// TIA Portal V19 export
VAR_GLOBAL   // PLC tag table "Default tag table"
   "CPU RUN" AT %I0.0 : Bool;
   "SPARE(1)" AT %I0.1 : Bool;
   "SPARE(2)" AT %I0.2 : Bool;
   "P-201 A RO 1 FEED PUMP TRIP" AT %I0.3 : Bool;
   "P-201 B RO 1 FEED PUMP TRIP" AT %I0.4 : Bool;
   "P-201 C RO 1 FEED PUMP TRIP" AT %I0.5 : Bool;
   "P-301 A RO 1 HPP PUMP TRIP" AT %I0.6 : Bool;
   "P-301 B RO B HPP PUMP TRIP" AT %I0.7 : Bool;
   "P-401 A RO 2 FEED PUMP TRIP" AT %I1.0 : Bool;
   "P-401 B RO 2 FEED PUMP TRIP" AT %I1.1 : Bool;
   "P-401 C RO 2 FEED PUMP TRIP" AT %I1.2 : Bool;
   "P 401 A RO 2 HPP PUMP TRIP" AT %I1.3 : Bool;
   "P-401 B RO 2 HPP PUMP TRIP" AT %I1.4 : Bool;
   "LPS 301 RO 1" AT %I1.5 : Bool;
   "P-202 A RO 1 FEED PUMP" AT %Q0.0 : Bool;
   "P-202 B RO 1 FEED PUMP" AT %Q0.1 : Bool;
   "P-202 C RO 1 FEED PUMP" AT %Q0.2 : Bool;
   "P-301 A RO 1 HPP PUMP" AT %Q0.3 : Bool;
   "P-301 B RO 1 HPP PUMP" AT %Q0.4 : Bool;
   "P-401 A RO 2 FEED PUMP" AT %Q0.5 : Bool;
   "P-401 B RO 2 FEED PUMP" AT %Q0.6 : Bool;
   "P-401 C RO 2 FEED PUMP" AT %Q0.7 : Bool;
   "P-402  A RO 2 HPP" AT %Q1.0 : Bool;
   "P-402 B" AT %Q1.1 : Bool;
   "HPS-301 RO 1 PRESSURE SWITCH" AT %I8.0 : Bool;
   "LPS-302 RO 1 PRESSURE SWITCH" AT %I8.1 : Bool;
   "HPS-302 RO 1 PRESSURE SWITCH" AT %I8.2 : Bool;
   "LPS-401 RO 2 PRESSURE SWITCH" AT %I8.3 : Bool;
   "HPS-401 RO 2 PRESSURE SWITCH" AT %I8.4 : Bool;
   "LPS-402 RO 2 PRESSURE SWITCH" AT %I8.5 : Bool;
   "HPS-402 RO 2 PRESSURE SWITCH" AT %I8.6 : Bool;
   "DP-703 RO 1 DOSER LEVEL SWITCH" AT %I8.7 : Bool;
   "DP-704 RO 1 DOSER LEVEL SWITCH" AT %I9.0 : Bool;
   "DP-705 RO 1 DOSER LEVEL SWITCH" AT %I9.1 : Bool;
   "P-501 A EDI FEED PUMP TRIP" AT %I9.2 : Bool;
   "P-501 B EDI FEED PUMP TRIP" AT %I9.3 : Bool;
   "P-501 C EDI FEED PUMP TRIP" AT %I9.4 : Bool;
   "EDI 501 A TRIP" AT %I9.5 : Bool;
   "EDI 501 B TRIP" AT %I9.6 : Bool;
   "P-501 A EDI FEED PUMP" AT %Q8.0 : Bool;
   "P-501 B EDI FEED PUMP" AT %Q8.1 : Bool;
   "P-501 C EDI FEED PUMP" AT %Q8.2 : Bool;
   "EDI 501" AT %Q8.3 : Bool;
   "EDI 502" AT %Q8.4 : Bool;
   "DP 703" AT %Q8.5 : Bool;
   "DP 704" AT %Q8.6 : Bool;
   "DP 705" AT %Q8.7 : Bool;
   "ABV 301" AT %Q9.0 : Bool;
   "ABV 302" AT %Q9.1 : Bool;
   "AGLV-301" AT %Q9.2 : Bool;
   "AGLV-302" AT %Q9.3 : Bool;
   "AGLV-401" AT %Q9.4 : Bool;
   "AGLV-402" AT %Q9.5 : Bool;
   "AGLV-501" AT %Q9.6 : Bool;
   "AGLV-502" AT %Q9.7 : Bool;
   "P-201 A RO 1 FEED PUMP FEED BACK" AT %I12.0 : Bool;
   "P-201 B RO 1 FEED PUMP FEED BACK" AT %I12.1 : Bool;
   "P-201 C RO 1 FEED PUMP FEED BACK" AT %I12.2 : Bool;
   "P-301 A RO 1 HPP PUMP FEED BACK" AT %I12.3 : Bool;
   "P-301 B RO 1 HPP PUMP FEED BACK" AT %I12.4 : Bool;
   "P-401 A R0 2 FEED PUMP FEED BACK" AT %I12.5 : Bool;
   "P-401 B RO 2 FEED PUMP FEED BACK" AT %I12.6 : Bool;
   "P-401 C RO 2 FEED PUMP FEED BACK" AT %I12.7 : Bool;
   "P-402 A RO 2 HPP PUMP FEED BACK" AT %I13.0 : Bool;
   "P-402 B RO 2 HPP PUMP FEED BACK" AT %I13.1 : Bool;
   "P-501 A EDI FEED PUMP FEED BACK" AT %I13.2 : Bool;
   "P-501 B EDI FEED PUMP FEED BACK" AT %I13.3 : Bool;
   "P-501 C EDI FEED PUMP FEED BACK" AT %I13.4 : Bool;
   "SPARE(3)" AT %I13.5 : Bool;
   "ABFV-301 FEED BACK OPEN" AT %I13.6 : Bool;
   "ABFV-301 FEED BACK CLOSE" AT %I13.7 : Bool;
   "ABFV-302 OPEN FEED BACK" AT %I16.0 : Bool;
   "ABFV-302 CLOSE FEED BACK" AT %I16.1 : Bool;
   "AGLV-301 OPEN FEED BACK" AT %I16.2 : Bool;
   "AGLV-301 CLOSE FEED BACK" AT %I16.3 : Bool;
   "AGLV-302 OPEN FEED BACK" AT %I16.4 : Bool;
   "AGLV-302 CLOSE FEED BACK" AT %I16.5 : Bool;
   "AGLV-401 OPEN FEED BACK" AT %I16.6 : Bool;
   "AGLV-401 CLOSE FEED BACK" AT %I16.7 : Bool;
   "AGLV-402 OPEN FEED BACK" AT %I17.0 : Bool;
   "AGLV-402 CLOSE FEED BACK" AT %I17.1 : Bool;
   "AGLV-501OPEN FEED BACK" AT %I17.2 : Bool;
   "AGLV-501 CLOSE FEED BACK" AT %I17.3 : Bool;
   "AGLV-502 OPEN FEED BACK" AT %I17.4 : Bool;
   "AGLV-502 CLOSE FEED BACK" AT %I17.5 : Bool;
   "SPARE(4)" AT %I17.6 : Bool;
   "SPARE(5)" AT %I17.7 : Bool;
   "OXIDATION REDUCTION POTENTIO METER 301" AT %IW144 : Int;
   "CONDUCTIVITY INDUCTOR CUM TRANSMITTER 301" AT %IW146 : Int;
   "PH INDICATOR CUM TRANSMITTER 301" AT %IW148 : Int;
   "PH INDICATOR CUM TRANSMITTER 302" AT %IW150 : Int;
   "CONDUCTIVITY INDICATOR CUM TRANSMITTER 302" AT %IW152 : Int;
   "LEVEL TRANSMITTER 401" AT %IW154 : Int;
   "PH INDICATOR CUM TRANSMITTER 401" AT %IW156 : Int;
   "CONDUCTIVITY INDICATOR CUM TRANSMITTER 401" AT %IW158 : Int;
   "CONFUCTIVITY INDICATOR CUM TRANSMITTER 402" AT %IW160 : Int;
   "PH INDICATOR CUM TRANSMITTER 402" AT %IW162 : Int;
   "LEVEL TRANSMITTER 501" AT %IW164 : Int;
   "FLOW INDICATOR TOTALOZER 501" AT %IW166 : Int;
   "PRESSURE TRANSMITTER 501" AT %IW168 : Int;
   "FLOW INDICATOR TRANSMITTER 502" AT %IW170 : Int;
   "PRESSURE TRANSMITTER 502" AT %IW172 : Int;
   "PRESSURE TRANSMITTER 503" AT %IW174 : Int;
   "PRESSURE TRANSMITTER 504" AT %IW176 : Int;
   "PRESSURE TRANSMITTER 505" AT %IW178 : Int;
   "PRESSURE TRANSMITTER 506" AT %IW180 : Int;
   "PH INDICATOR CUM TRANSMITTER 501" AT %IW182 : Int;
   "PH INDICATOR CUM TRANSMITTER 502" AT %IW184 : Int;
   "RESISTIVITY CUM TRANSMITTER 501" AT %IW186 : Int;
   "RESISTIVITY CUM TRANSMITTER 502" AT %IW188 : Int;
   "LEVEL TRANSMITTER 502" AT %IW190 : Int;
   "FLOW INDICATOR TRANSMITTER 503" AT %IW192 : Int;
   "FLOW INDICATOR TRANSMITTER 504" AT %IW194 : Int;
   "FLOW INDICATOR TRANSMITTER 505" AT %IW196 : Int;
   "FLOW INDICATOR TRANSMITTER 506" AT %IW198 : Int;
   "FLOW INDICATOR TRANSMITTER 507" AT %IW200 : Int;
   "FLOW INDICATOR TRANSMITTER 508" AT %IW202 : Int;
   "SPARE(6)" AT %IW204 : Int;
   "SPARE(7)" AT %IW206 : Int;
   "SPARE(8)" AT %I9.7 : Bool;
   Tag_1 AT %Q1.2 : Bool;
   Tag_2 AT %I1.6 : Bool;
   Clock_Byte AT %MB0 : Byte;
   Clock_10Hz AT %M0.0 : Bool;
   Clock_5Hz AT %M0.1 : Bool;
   "Clock_2.5Hz" AT %M0.2 : Bool;
   Clock_2Hz AT %M0.3 : Bool;
   "Clock_1.25Hz" AT %M0.4 : Bool;
   Clock_1Hz AT %M0.5 : Bool;
   "Clock_0.625Hz" AT %M0.6 : Bool;
   "Clock_0.5Hz" AT %M0.7 : Bool;
   System_Byte AT %MB1 : Byte;
   FirstScan AT %M1.0 : Bool;
   DiagStatusUpdate AT %M1.1 : Bool;
   AlwaysTRUE AT %M1.2 : Bool;
   AlwaysFALSE AT %M1.3 : Bool;
   "PLC_2 HOOTER" AT %M2.0 : Bool;
   "SET TIME" AT %MW4 : Int;
   "LT 201" AT %MD6 : Real;
   TAG122 AT %M2.1 : Bool;
   TEST_1 AT %M2.2 : Bool;
   TEST_2 AT %M2.3 : Bool;
   TEST_3 AT %M2.4 : Bool;
   GGG AT %M2.5 : Bool;
   GGG1 AT %M2.6 : Bool;
   HH AT %M2.7 : Bool;
   HOOTER AT %M3.0 : Bool;
   QQQ AT %M3.1 : Bool;
   YYU AT %M3.2 : Bool;
   YYY1 AT %M3.3 : Bool;
   YYY2 AT %M3.4 : Bool;
   SLAVE1_WRITE_DONE AT %M3.5 : Bool;
   SLAVE1_WRITE_BUSY AT %M3.6 : Bool;
   SLAVE1_WRITE_ERROR AT %M3.7 : Bool;
   CYCLE AT %MW10 : Int;
   HHH AT %M12.0 : Bool;
   Tag_3 AT %IW64 : Int;
   Tag_4 AT %IW100 : Int;
   KKKK AT %MW14 : Int;
   KKK AT %M12.1 : Bool;
   JJJJ AT %M12.2 : Bool;
   hvvvvhh AT %M12.3 : Bool;
   kkkkk AT %M12.4 : Bool;
   FFF AT %M12.5 : Bool;
   FFF1 AT %M12.6 : Bool;
END_VAR
